// TIA Portal V20 export
FUNCTION_BLOCK "Simulation"   // FB50061, LAD
// stored: MemoryReserve 100, Namespace Unit1.Em6, SetENOAutomatically false
   VAR_INPUT
      simulation { ExternalAccessible := 'False'; ExternalVisible := 'False'; ExternalWritable := 'False'} : Bool;
   END_VAR
   VAR
      instActuator { ExternalAccessible := 'False'; ExternalVisible := 'False'; ExternalWritable := 'False'} : Array[0..9] of "LER_SimActuator";
   END_VAR
BEGIN

REGION Network 1: Two Way Actuator
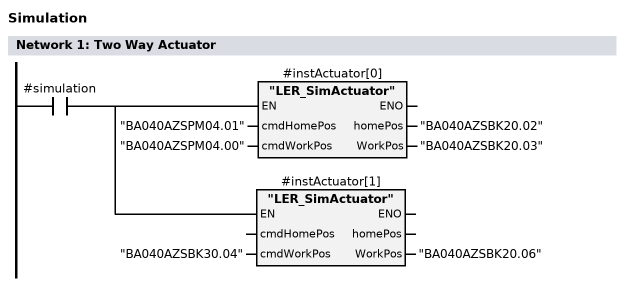
   RUNG wire#powerrail
      Contact( #simulation )
      wire#w1
      #instActuator[0](cmdHomePos := "BA040AZSPM04.01", cmdWorkPos := "BA040AZSPM04.00", homePos => "BA040AZSBK20.02", WorkPos => "BA040AZSBK20.03")
   END_RUNG
   RUNG wire#w1
      #instActuator[1](cmdHomePos :=, cmdWorkPos := "BA040AZSBK30.04", homePos =>, WorkPos => "BA040AZSBK20.06")
   END_RUNG
   // the same network as SCL:
   IF #simulation THEN
       #instActuator[0](cmdHomePos := "BA040AZSPM04.01",   // "LER_SimActuator"
                        cmdWorkPos := "BA040AZSPM04.00",
                        homePos => "BA040AZSBK20.02",
                        WorkPos => "BA040AZSBK20.03");
       #instActuator[1](cmdWorkPos := "BA040AZSBK30.04", WorkPos => "BA040AZSBK20.06");   // "LER_SimActuator"
   END_IF;
END_REGION
END_FUNCTION_BLOCK
